// TIA Portal V19 export
TYPE "C904_VAR_IF_SPI_TYPIC"
   STRUCT
      WRE { ExternalAccessible := 'False'; ExternalVisible := 'False'; ExternalWritable := 'False'} : USInt;   // Actueel actief regime
      BMO_HAND { ExternalAccessible := 'False'; ExternalVisible := 'False'; ExternalWritable := 'False'} : Bool;   // TRUE = Regime handmatig ingesteld via lokale bediening
      STO { ExternalAccessible := 'False'; ExternalVisible := 'False'; ExternalWritable := 'False'} : Struct   // Opsomming van alle storingen
         A001 : Bool;   // Beveiliging aangesproken
         A002 : Bool;   // Beveiliging No-Break aangesproken
         A003 : Bool;   // Overspanningsbeveiliging aangesproken
         A004 : Bool;   // Schuif ALSB uitgeschakeld
         A005 : Bool;   // Schuif ALSB in test
         A006 : Bool;   // Schuif ALSB uitgereden
         A007 : Bool;   // Nisdeur niet gesloten
         A008 : Bool;   // Storing tracing
      END_STRUCT;
   END_STRUCT;
END_TYPE
